{attribute 'GeneratedUsingTerminal: BK1120-0000-0020'}
{attribute addProperty BoxType "BK1120-0000-0020"}
{attribute addProperty Id "Term_380_KL1002KL1002_BB38DA8F0"}
{attribute addProperty CRC "1642230361"}
{attribute addProperty Size "0"}
TYPE A_0007_BK1120_0000_0020_61E27259 EXTENDS BK1120_A2FCADE7 :
STRUCT
	{attribute addProperty Name "Term_380_KL1002"}
	Term_380_KL1002 : KL1002_BB38DA8F;
END_STRUCT
END_TYPE

(* stored: Version 1.2.0.0, ProductVersion 3.1.4024.9
   DUT A_0007_BK1120_0000_0020_61E27259: Id {f44c2e97-92bb-4bbe-95cc-8a3ba7577297} *)
